(* IEC 61131-3 sources: RL_MAR/experiments/comparison/llm4plc/results/gpt-4o_20260507_114630/20260507_121016, 3 files *)

(* ---- generated_code_iteration_0.st ---- *)
plaintext
START_ST
FUNCTION_BLOCK FB_Sum
VAR_INPUT
    maxValue : INT; // Specifies the maximum value for the summation loop
END_VAR

VAR_OUTPUT
    wData : WORD; // Stores the sum of integers from 0 to maxValue
END_VAR

VAR
    II : INT; // Loop index variable
    state : INT; // State variable to track the current state
    prevState : INT; // Previous state variable (optional, for debugging or tracking purposes)
END_VAR

// State Definitions
// STATE 0: INITIALIZE
// STATE 1: SUMMATION LOOP
// STATE 2: COMPLETION

// Initialization of the function block
IF state = 0 THEN
    // STATE 0: INITIALIZE
    wData := 0; // Initialize wData to 0
    II := 0; // Initialize loop index to 0
    prevState := state; // Update previous state
    state := 1; // Transition to STATE 1 (Summation Loop)
ELSIF state = 1 THEN
    // STATE 1: SUMMATION LOOP
    wData := wData + WORD(II); // Add the current value of II to wData
    II := II + 1; // Increment the loop index
    IF II > maxValue THEN
        prevState := state; // Update previous state
        state := 2; // Transition to STATE 2 (Completion)
    END_IF;
ELSIF state = 2 THEN
    // STATE 2: COMPLETION
    // No further operations; remain in this state indefinitely
    prevState := state; // Update previous state
    // wData holds the final summation result
END_IF;

END_FUNCTION_BLOCK
END_ST

(* ---- generated_code_iteration_1.st ---- *)
START_REASON
The validation feedback indicates that the issue lies with the use of `WORD(II)` in the summation operation. The CODESYS compiler expects a semicolon (`;`) instead of `WORD`. This suggests that the explicit type conversion `WORD(II)` is either incorrect or not supported in this context. To resolve this, I will replace `WORD(II)` with a valid operation or type conversion that adheres to CODESYS standards. Additionally, I will ensure the code is syntactically correct and logically sound.
END_REASON

START_ST
FUNCTION_BLOCK FB_Sum
VAR_INPUT
    maxValue : INT; // Specifies the maximum value for the summation loop
END_VAR

VAR_OUTPUT
    wData : WORD; // Stores the sum of integers from 0 to maxValue
END_VAR

VAR
    II : INT; // Loop index variable
    state : INT; // State variable to track the current state
    prevState : INT; // Previous state variable (optional, for debugging or tracking purposes)
END_VAR

// State Definitions
// STATE 0: INITIALIZE
// STATE 1: SUMMATION LOOP
// STATE 2: COMPLETION

// Initialization of the function block
IF state = 0 THEN
    // STATE 0: INITIALIZE
    wData := 0; // Initialize wData to 0
    II := 0; // Initialize loop index to 0
    prevState := state; // Update previous state
    state := 1; // Transition to STATE 1 (Summation Loop)
ELSIF state = 1 THEN
    // STATE 1: SUMMATION LOOP
    wData := wData + WORD_TO_WORD(II); // Correct type conversion for summation
    II := II + 1; // Increment the loop index
    IF II > maxValue THEN
        prevState := state; // Update previous state
        state := 2; // Transition to STATE 2 (Completion)
    END_IF;
ELSIF state = 2 THEN
    // STATE 2: COMPLETION
    // No further operations; remain in this state indefinitely
    prevState := state; // Update previous state
    // wData holds the final summation result
END_IF;

END_FUNCTION_BLOCK
END_ST

(* ---- generated_code_iteration_2.st ---- *)
START_REASON
The validation feedback indicates that the issue lies in the summation operation `wData := wData + WORD_TO_WORD(II);`. The error message suggests that the type conversion `WORD_TO_WORD(II)` is invalid or not supported in this context. Additionally, it appears that the addition operation is causing a type mismatch because `wData` is of type `WORD`, and `II` is of type `INT`.

To resolve this, I will:
1. Ensure proper type conversion between `INT` and `WORD`. Specifically, I will use `TO_WORD(II)` instead of `WORD_TO_WORD(II)` as it is the correct function for converting an `INT` to a `WORD` in CODESYS.
2. Verify that the addition operation is valid by ensuring that both operands are of the same type (`WORD`).
3. Ensure that the code adheres to CODESYS standards and compiles without errors.

I will now update the code to address these issues.
END_REASON

START_ST
FUNCTION_BLOCK FB_Sum
VAR_INPUT
    maxValue : INT; // Specifies the maximum value for the summation loop
END_VAR

VAR_OUTPUT
    wData : WORD; // Stores the sum of integers from 0 to maxValue
END_VAR

VAR
    II : INT; // Loop index variable
    state : INT; // State variable to track the current state
    prevState : INT; // Previous state variable (optional, for debugging or tracking purposes)
    tempSum : INT; // Temporary variable to store the summation result as INT
END_VAR

// State Definitions
// STATE 0: INITIALIZE
// STATE 1: SUMMATION LOOP
// STATE 2: COMPLETION

// Initialization of the function block
IF state = 0 THEN
    // STATE 0: INITIALIZE
    tempSum := 0; // Initialize tempSum to 0
    II := 0; // Initialize loop index to 0
    prevState := state; // Update previous state
    state := 1; // Transition to STATE 1 (Summation Loop)
ELSIF state = 1 THEN
    // STATE 1: SUMMATION LOOP
    tempSum := tempSum + II; // Add the current loop index to tempSum
    II := II + 1; // Increment the loop index
    IF II > maxValue THEN
        prevState := state; // Update previous state
        state := 2; // Transition to STATE 2 (Completion)
    END_IF;
ELSIF state = 2 THEN
    // STATE 2: COMPLETION
    wData := TO_WORD(tempSum); // Convert the final summation result to WORD and store in wData
    prevState := state; // Update previous state
    // No further operations; remain in this state indefinitely
END_IF;

END_FUNCTION_BLOCK
END_ST
